TYPE ST145_Feeder_e : ST110_Feeder_e;
END_TYPE

(* stored: Version 1.1.0.1, ProductVersion 3.1.4024.6
   DUT ST145_Feeder_e: Id {7b2bc12b-1d43-4d92-933f-fc5ab7037521} *)
